// TIA Portal V18 export
FUNCTION_BLOCK "encoder2"   // FB62, FBD
{ S7_Optimized_Access := 'TRUE' }
VERSION : 0.1
// stored: AutoNumber true, IsIECCheckEnabled false, IsRetainMemResEnabled false, MemoryReserve 100, SetENOAutomatically false, UDAEnableTagReadback false
   VAR_INPUT
      xCal : Bool;
      ENC : Real;
      posCal : Real;
   END_VAR
   VAR_OUTPUT
      i_times_cal : Int;
      retain_test : Bool;
      POS : Real;
   END_VAR
   VAR
      xCal_filtered : Bool;
      not_first_scan : Bool;
      offset : Real;
   END_VAR
   VAR RETAIN
      MEM : Real;
   END_VAR
   VAR
      xCal_mem : Bool;
   END_VAR
   VAR RETAIN
      calibrated : Bool;
   END_VAR
   VAR
      ton_block_calib { S7_SetPoint := 'True'} : TON_TIME;
      tonFilter { S7_SetPoint := 'True'} : TON_TIME;
   END_VAR
BEGIN

REGION Network 1
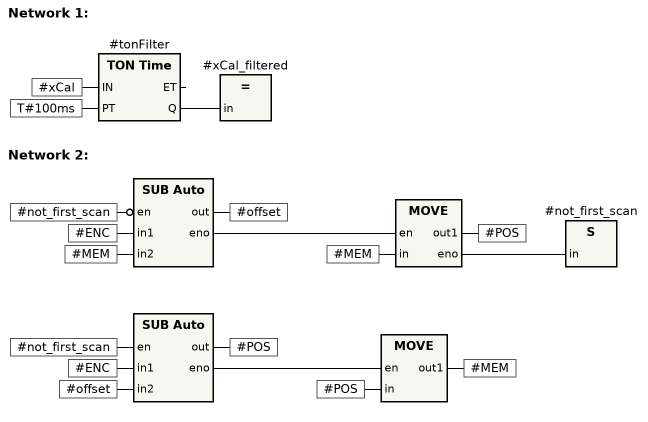
   #tonFilter(IN := #xCal, PT := T#100ms);   // TON
   #xCal_filtered := #tonFilter.Q;
END_REGION

REGION Network 2
   IF NOT #not_first_scan THEN
       #offset := #ENC - #MEM;
       #POS := #MEM;
       #not_first_scan := TRUE;
   END_IF;
   IF #not_first_scan THEN
       #POS := #ENC - #offset;
       #MEM := #POS;
   END_IF;
END_REGION

REGION Network 3 (SCL)
   IF #xCal_filtered AND NOT #xCal_mem THEN
       #offset := #ENC - #posCal;
       #calibrated := true;
       #i_times_cal := #i_times_cal + 1;
   END_IF;
   #xCal_mem := #xCal_filtered;
END_REGION
END_FUNCTION_BLOCK
